TYPE ST_SafetyOutputGroup :
STRUCT
	iGroupNumber : INT;
	aSafetyOuputs : ARRAY[1..GVL_Safety.nSAFETY_OUTPUTS] OF BOOL;
END_STRUCT
END_TYPE

(* stored: Version 1.1.0.1, ProductVersion 3.1.4024.11
   DUT ST_SafetyOutputGroup: Id {f4256feb-14ff-44b1-bf30-19175d40816f} *)
